FUNCTION_BLOCK dummy_cap_fb (* FB for testing N vars *)
  (* Standard: 61499-2 *)
  (* Version 1.0, 2025-05-16, Test *)
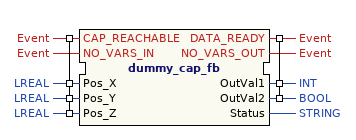
  EVENT_INPUT
    CAP_REACHABLE WITH Pos_X, Pos_Y, Pos_Z;
    NO_VARS_IN;
  END_EVENT
  EVENT_OUTPUT
    DATA_READY WITH OutVal1, OutVal2;
    NO_VARS_OUT;
  END_EVENT
  VAR_INPUT
    Pos_X : LREAL;
    Pos_Y : LREAL;
    Pos_Z : LREAL;
  END_VAR
  VAR_OUTPUT
    OutVal1 : INT;
    OutVal2 : BOOL;
    Status : STRING;
  END_VAR
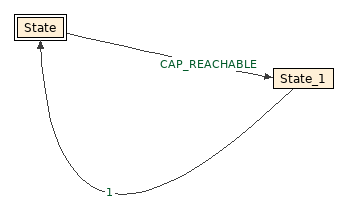
  EC_STATES
    State;
    State_1;
  END_STATES
  EC_TRANSITIONS
    State TO State_1 := CAP_REACHABLE;
    State_1 TO State := 1;
  END_TRANSITIONS
END_FUNCTION_BLOCK
